INTERFACE I_Module EXTENDS I_Element

METHOD PUBLIC M_Mode : BOOL
VAR_INPUT
	eMode:		E_Mode;
END_VAR
END_METHOD

PROPERTY PUBLIC P_Mode : E_Mode
GET
END_GET
END_PROPERTY

END_INTERFACE

(* stored: Version 1.1.0.1
   Itf I_Module: Id {17c5a5c0-e93a-0aed-1dd7-b12ea548c450}
   Method M_Mode: Id {208c4c43-a103-0c2c-0258-2704597726e6}
   Property P_Mode: Id {e048b2ce-4d45-02c7-3379-8e81d7ba5300}
   Get Get: Id {ee8b9205-2345-0b77-239a-ffedae0545c4} *)
